Fanuc KAREL source: kt00193.compact.KL

PROGRAM KT00193
%STACKSIZE=65535
%PRIORITY=65535
%NOLOCKGROUP
VAR
B1 : BOOLEAN
B2 : BOOLEAN
OUT : BOOLEAN
BEGIN
B1=TRUE
B2=FALSE
B1=TRUE
B2=FALSE
OUT=(B1 AND B2)
END KT00193
